// TIA Portal V20 export
TYPE "IO_MOT"
   STRUCT
      IN { ExternalAccessible := 'False'; ExternalVisible := 'False'; ExternalWritable := 'False'} : Struct
         Trip : Bool;
         FwdFb : Bool;
         RevFb : Bool;
      END_STRUCT;
      OUT { ExternalAccessible := 'False'; ExternalVisible := 'False'; ExternalWritable := 'False'} : Struct
         FwdCmd : Bool;
         RevCmd : Bool;
      END_STRUCT;
   END_STRUCT;
END_TYPE
